(* PLC project  *)

CONFIGURATION FSOE_AxisMR
END_CONFIGURATION
